ABB RobotStudio station: Tp2_20201212-015021.rsstn

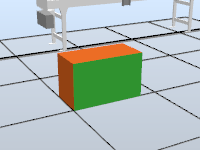
Station Tp2 (saved by RobotStudio 20.1.8982.0)
Layout (positions relative to the parent item):
  - IRB660_180_315__01 [mechanism, from Robots\IRB660_180_315__01.rslib] at (0, 0, 0) mm; joint values [0.0199, 0, 0, 0] (rad or m)
  - 400_guide [part, from Equipment\Conveyor Guide 400.rslib] at (0, 1500, 0) mm, rotated rx 0 ry 0 rz 90 deg
  - Euro Pallet [graphiccomponentgroup, from Equipment\Euro Pallet.rslib] at (1000, -1425, 435) mm
    - Body 1 [part, from Equipment\Euro Pallet.rslib]
  - 950_4000_h2_2 [part, from Equipment\Conveyor 950 4000 h2.rslib] at (1000, -1500, 0) mm
  - Pieza_2 [part]
  - topePallet [frame] at (1000, -1025, 435) mm
  - basePallet [frame] at (1000, -1025, 435) mm
  - topeCajas [frame] at (-240, 1500, 770) mm, rotated rx 0 ry 0 rz 90 deg
Attachment: Euro Pallet is attached to 950_4000_h2_2
Attachment: basePallet is attached to Euro Pallet
Attachment: topePallet is attached to 950_4000_h2_2
Attachment: topeCajas is attached to 400_guide
